SUBAPPLICATION Softkey_Aux_IXA_TO_Remote_WRITE (* VT-SoftKey lesen ODER AUX-Zuweisung (Joystick) lesen ODER lokaler Web-Override (z.B. vt-ui-mirror auf demselben Modul) + Remote-OPC-UA-Write an Zielmodul (generisch, ein Kanal, ohne Status-Feedback) *)
  (* Standard: 61499-2; Description: Copyright (c) 2026 Meisterschulen am Ostbahnhof This program and the accompanying materials are made available under the terms of the Eclipse Public License 2.0 which is available at https://www.eclipse.org/legal/epl-2.0/ SPDX-License-Identifier: EPL-2.0 *)
  (* Version 1.0, 2026-09-07, Franz Höpfinger, Meisterschulen am Ostbahnhof, Aus Softkey_Aux_IXA_TO_Remote_WRITE_BG_OPC herausgeloest: nur die Kommando-Seite (Quellen-ODER + Remote-Write), ohne Status-Feedback *)
  PACKAGE MyLib::sys;
  IMPORT isobus::UT::Q::const::IDs::ID_NULL;
  (* Documentation:
  SoftKey UND Aux → Remote-OPC-UA-Write (nur Kommando, kein Status)
   Kommando-Haelfte von Softkey_Aux_IXA_TO_Remote_WRITE_BG_OPC, herausgeloest als eigener Baustein: SoftKey (u16ObjId), Aux-Zuweisung (u16ObjIdA) und ein lokaler Web-Override (ID_WEB_READ) werden per AX_OR_3 zusammengefuehrt und per AX_CLIENT_1_0 (ID_WRITE_REMOTE) ans Zielmodul geschrieben.
   Kein Status-Feedback/Hintergrundfarbe hier - dafuer AX_SUBSCRIBE_BG3_WEB_OPC danebenstellen (gleiche u16ObjId/u16ObjIdA-Werte durchreichen). Fuer die komplette, vorverdrahtete Kombination beider Bausteine weiterhin Softkey_Aux_IXA_TO_Remote_WRITE_BG_OPC verwenden.
  *)
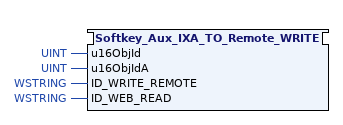
  VAR_INPUT
    u16ObjId : UINT := ID_NULL; (* Object ID SoftKey (VT) *)
    u16ObjIdA : UINT := ID_NULL; (* Object ID AuxFunction2 (VT) *)
    ID_WRITE_REMOTE : WSTRING; (* Remote-Write-Adresse zum Zielmodul (Befehl, ACTION=WRITE, CLIENT) *)
    ID_WEB_READ : WSTRING; (* Lokale Subscribe-Adresse fuer einen Web-Client (z.B. vt-ui-mirror) auf demselben Modul, ODER-verknuepft mit SoftKey und AUX *)
  END_VAR
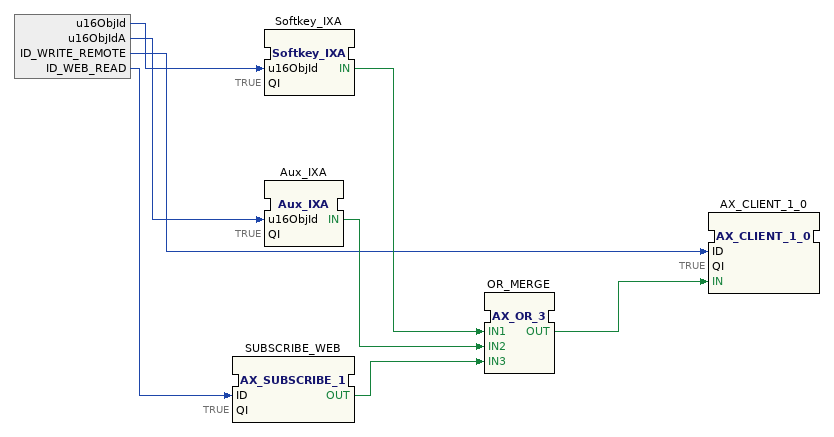
  FBS
    Softkey_IXA : isobus::UT::io::Softkey::Softkey_IXA(QI := TRUE);
    Aux_IXA : isobus::UT::io::Auxiliary::IN::Aux_IXA(QI := TRUE);
    SUBSCRIBE_WEB : adapter::net::AX_SUBSCRIBE_1(QI := TRUE);
    OR_MERGE : adapter::booleanOperators::AX_OR_3;
    AX_CLIENT_1_0 : adapter::net::AX_CLIENT_1_0(QI := TRUE);
  END_FBS
  DATA_CONNECTIONS
    u16ObjId TO Softkey_IXA.u16ObjId;
    u16ObjIdA TO Aux_IXA.u16ObjId;
    ID_WEB_READ TO SUBSCRIBE_WEB.ID;
    ID_WRITE_REMOTE TO AX_CLIENT_1_0.ID;
  END_CONNECTIONS
  ADAPTER_CONNECTIONS
    Softkey_IXA.IN TO OR_MERGE.IN1;
    Aux_IXA.IN TO OR_MERGE.IN2;
    SUBSCRIBE_WEB.OUT TO OR_MERGE.IN3;
    OR_MERGE.OUT TO AX_CLIENT_1_0.IN;
  END_CONNECTIONS
END_SUBAPPLICATION
